{attribute 'qualified_only'}
VAR_GLOBAL
    (*******************************************************************)
    (* Allgemeine Globale Variablen *)
    (*******************************************************************)
    (******* FREIGABEN *********)
    //ST01
    xFG_ST01akVZ : BOOL; // Vereinzelung Teil anwesend
    xFG_ST01akWT : BOOL; // WT anwesend
    //ST02
    xFG_ST02akWT : BOOL; // WT anwesend

    st105_aut : FB_AUT_105;   // Laden Filtergehäuse
    st110_aut : FB_AUT_110;    // Laden RFID-Ring
    st115_aut : FB_AUT_115;    // Laden kristal
    st120_aut : FB_AUT_120;    // Laden Solerohr
    st125_aut : FB_AUT_125;    // Laden filterhut
    st130_aut : FB_AUT_130;    // Dosieren A
    st135_aut : FB_AUT_MODIFY; // Dosieren B
    st140_aut : FB_AUT_MODIFY; // Niveaukontrolle
    st145_aut : FB_AUT_145;    // Laden Patronendeckel
    st150_aut : FB_AUT_MODIFY; // Utralson A
    st155_aut : FB_AUT_MODIFY; // Ultrason B
    st160_aut : FB_AUT_MODIFY; // Prüfig A
    st165_aut : FB_AUT_MODIFY; // Prüfig B
    st170_aut : FB_AUT_MODIFY; // Program RFID
    st175_aut : FB_AUT_MODIFY; // Laser A
    st176_aut : FB_AUT_MODIFY; // Laser B
    st180_aut : FB_AUT_180;    // Entladen schlecht
    st185_aut : FB_AUT_185;    // Entladen gut
    st1xx_aut : FB_AUT_175;    // test laser trumpf

END_VAR

(* stored: Version 1.1.0.1, ProductVersion 3.1.4024.6
   GVL GVL: Id {94734850-411d-4576-a0e7-f0a38cdbbc44} *)
